TYPE DUT_Statistics :
STRUCT
	OEE_Enable				: BOOL;
	OEE_Reset				: BOOL;
END_STRUCT
END_TYPE

(* stored: Version 1.1.0.1, ProductVersion 3.1.4024.13
   DUT DUT_Statistics: Id {e471b8b5-6b6b-4915-953b-204eac4ab1a1} *)
